// TwinCAT 3 PLC project UnitTests
// Title: tcl_StringUtils_UnitTests
// Company: Red Rock Controls Limited
// Author: Roger Christopher
// ProjectVersion: 1.0.1.0
// Description: Tests tcl_StringUtils V 1.0.5.0 Updated to use tcl_SimpleUnitTestLibrary V1.0.2.0
// ProgramVersion: 3.1.4024.0
// libraries:
//   Tc2_Standard, * (Beckhoff Automation GmbH)
//   Tc2_System, * (Beckhoff Automation GmbH)
//   Tc2_Utilities, * (Beckhoff Automation GmbH)
//   Tc3_Module, * (Beckhoff Automation GmbH)
//   tcl_StringUtils, * (Red Rock Controls Limited)
//   tcl_UnitTestLibrary, * (Red Rock Controls Limited)
// project tree:
//   / PlcTask.TcTTO
//   Unit Tests/ MAIN.TcPOU, T_TestSuite.TcPOU
//   Unit Tests/String Utils/Conversion/ Test_StringToIpAddress.TcPOU
//   Unit Tests/String Utils/Date Time Formatting Tests/ Test_F_DateAsString_ReturnsDateString.TcPOU, Test_F_DateTimeAsString.TcPOU, Test_F_DateTimeAsString_ms.TcPOU, Test_F_TimeAsString_Returns24HourFormat.TcPOU, Test_F_TimeAsString_ReturnsLeadingZeros.TcPOU, Test_F_TimeAsString_ms_ReturnsString_ms.TcPOU, Test_F_TimestampAsFilename_ReturnsValue.TcPOU, Test_F_TimestampAsFilename_ms.TcPOU
//   Unit Tests/String Utils/Format String Tests/ Test_FormatStringWith4CharHexValue.TcPOU, Test_FormatStringWith8CharHexValue.TcPOU, Test_F_PadString_PadsShortStrings.TcPOU, Test_F_PadString_TruncsLongStrings.TcPOU
//   Unit Tests/String Utils/LTrimEx/ Test_LTrimEx_HandlesEmptySubject.TcPOU, Test_LTrimEx_HandlesTrimmingManyChars.TcPOU, Test_LTrimEx_HandlesTrimmingNoChars.TcPOU
//   Unit Tests/String Utils/RTrimEx/ Test_RTrimEx_HandlesEmptySubject.TcPOU, Test_RTrimEx_HandlesTrimmingManyChars.TcPOU, Test_RTrimEx_HandlesTrimmingNoChars.TcPOU
//   Unit Tests/String Utils/String Split/ Test_TStringSplitter_Handles_Empty_String.TcPOU, Test_TStringSplitter_Handles_Empty_SubString.TcPOU, Test_TStringSplitter_Handles_Multiple_Empty.TcPOU, Test_TStringSplitter_ReturnsRemainder.TcPOU, Test_TStringSplitter_Splits_On_Tab.TcPOU
//   Unit Tests/String Utils/Trim/ Test_TrimEx_HandlesEmptySubject.TcPOU, Test_TrimEx_HandlesTrimmingOnlyWhitespace.TcPOU
// (motion and I/O tree: see PLC project tcl_stringutils)
// real-time tasks:
//   TASK PlcTask: cycle T#10ms, priority 1, ADS port 350

CONFIGURATION UnitTests
    RESOURCE PLC ON TwinCAT3
        TASK PlcTask(INTERVAL := T#10ms, PRIORITY := 1);
        PROGRAM MAIN WITH PlcTask : MAIN;
    END_RESOURCE
END_CONFIGURATION

// ---- Unit Tests/MAIN.TcPOU
PROGRAM MAIN
VAR
    TestSuite : T_TestSuite;
END_VAR

TestSuite();

END_PROGRAM

// ---- Unit Tests/T_TestSuite.TcPOU
{attribute 'call_after_init'}
FUNCTION_BLOCK T_TestSuite
VAR
    Test_StringToIpAddress                                 : Test_StringToIpAddress;
    Test_FormatStringWith4CharHexValue                     : Test_FormatStringWith4CharHexValue;
    Test_FormatStringWith8CharHexValue                     : Test_FormatStringWith8CharHexValue;
    Test_LTrimEx_HandlesEmptySubject                       : Test_LTrimEx_HandlesEmptySubject;
    Test_LTrimEx_HandlesTrimmingNoChars                    : Test_LTrimEx_HandlesTrimmingNoChars;
    Test_LTrimEx_HandlesTrimmingManyChars                  : Test_LTrimEx_HandlesTrimmingManyChars;
    Test_RTrimEx_HandlesEmptySubject                       : Test_RTrimEx_HandlesEmptySubject;
    Test_RTrimEx_HandlesTrimmingNoChars                    : Test_RTrimEx_HandlesTrimmingNoChars;
    Test_RTrimEx_HandlesTrimmingManyChars                  : Test_RTrimEx_HandlesTrimmingManyChars;
    Test_TrimEx_HandlesTrimmingOnlyWhitespace              : Test_TrimEx_HandlesTrimmingOnlyWhitespace;
    Test_TrimEx_HandlesEmptySubject                        : Test_TrimEx_HandlesEmptySubject;
    Test_F_DateAsString_ReturnsDateString                  : Test_F_DateAsString_ReturnsDateString;
    Test_F_DateTimeAsString_ReturnsDateTimeString          : Test_F_DateTimeAsString;
    Test_F_DateTimeAsString_ms_ReturnsDTStr                : Test_F_DateTimeAsString_ms;
    Test_F_TimeAsString_Returns24HourFormat                : Test_F_TimeAsString_Returns24HourFormat;
    Test_F_TimeAsString_ReturnsLeadingZeros                : Test_F_TimeAsString_ReturnsLeadingZeros;
    Test_F_TimeAsString_ms_ReturnsTimeString_ms            : Test_F_TimeAsString_ms_ReturnsString_ms;
    Test_F_TimestampAsFilenameString_ReturnsFilenameString : Test_F_TimestampAsFilename_ReturnsValue;
    Test_TStringSplitter_Handles_Empty_String              : Test_TStringSplitter_Handles_Empty_String;
    Test_TStringSplitter_ReturnsRemainder                  : Test_TStringSplitter_ReturnsRemainder;
    Test_TStringSplitter_Splits_On_Tab                     : Test_TStringSplitter_Splits_On_Tab;
    Test_TStringSplitter_Handles_Empty_SubString           : Test_TStringSplitter_Handles_Empty_SubString;
    Test_TStringSplitter_Handles_Multiple_Empty_SubStrings : Test_TStringSplitter_Handles_Multiple_Empty;
    Test_F_PadString_PadsShortStrings                      : Test_F_PadString_PadsShortStrings;
    Test_F_PadString_TruncsLongString                      : Test_F_PadString_TruncsLongStrings;
    Test_F_TimestampAsFilename_ms                          : Test_F_TimestampAsFilename_ms;
END_VAR

Test_StringToIpAddress.RunTest();
Test_FormatStringWith4CharHexValue.RunTest();
Test_FormatStringWith8CharHexValue.RunTest();
Test_LTrimEx_HandlesEmptySubject.RunTest();
Test_LTrimEx_HandlesTrimmingNoChars.RunTest();
Test_LTrimEx_HandlesTrimmingManyChars.RunTest();
Test_RTrimEx_HandlesEmptySubject.RunTest();
Test_RTrimEx_HandlesTrimmingNoChars.RunTest();
Test_RTrimEx_HandlesTrimmingManyChars.RunTest();
Test_TrimEx_HandlesTrimmingOnlyWhitespace.RunTest();
Test_TrimEx_HandlesEmptySubject.RunTest();
Test_F_DateAsString_ReturnsDateString.RunTest();
Test_F_DateTimeAsString_ReturnsDateTimeString.RunTest();
Test_F_DateTimeAsString_ms_ReturnsDTStr.RunTest();
Test_F_TimeAsString_Returns24HourFormat.RunTest();
Test_F_TimeAsString_ReturnsLeadingZeros.RunTest();
Test_F_TimeAsString_ms_ReturnsTimeString_ms.RunTest();
Test_F_TimestampAsFilenameString_ReturnsFilenameString.RunTest();
Test_TStringSplitter_Handles_Empty_String.RunTest();
Test_TStringSplitter_ReturnsRemainder.RunTest();
Test_TStringSplitter_Splits_On_Tab.RunTest();
Test_TStringSplitter_Handles_Empty_SubString.RunTest();
Test_TStringSplitter_Handles_Multiple_Empty_SubStrings.RunTest();
Test_F_PadString_PadsShortStrings.RunTest();
Test_F_PadString_TruncsLongString.RunTest();
Test_F_TimestampAsFilename_ms.RunTest();

END_FUNCTION_BLOCK

// ---- Unit Tests/String Utils/Conversion/Test_StringToIpAddress.TcPOU
FUNCTION_BLOCK Test_StringToIpAddress EXTENDS T_UnitTestBase
VAR
    SubjectString : T_MaxString := '192.168.1.120';
    Result        : ARRAY[1..4] OF BYTE;
END_VAR

{attribute 'analysis' := '-33'} // inhibit unused variable warning
METHOD RunTest
IF Retest THEN
	SUPER^.Init();
END_IF

IF TestCompleted THEN
	RETURN;
END_IF

Result := F_String_To_IPv4_Address(SubjectString);

AssertEquals_BYTE(Expected := 120,
                  Actual   := Result[1],
                  Message  := 'F_String_To_IPv4_Address(SubjectString)');

AssertEquals_BYTE(Expected := 1,
                  Actual   := Result[2],
                  Message  := 'F_String_To_IPv4_Address(SubjectString)');

AssertEquals_BYTE(Expected := 168,
                  Actual   := Result[3],
                  Message  := 'F_String_To_IPv4_Address(SubjectString)');

AssertEquals_BYTE(Expected := 192,
                  Actual   := Result[4],
                  Message  := 'F_String_To_IPv4_Address(SubjectString)');

TestCompleted := TRUE;
END_METHOD

END_FUNCTION_BLOCK

// ---- Unit Tests/String Utils/Format String Tests/Test_FormatStringWith4CharHexValue.TcPOU
FUNCTION_BLOCK Test_FormatStringWith4CharHexValue EXTENDS T_UnitTestBase
VAR_INPUT
END_VAR
VAR_OUTPUT
END_VAR
VAR
    FormattedString : T_MaxString;
    Value           : UINT;
END_VAR

{attribute 'analysis' := '-33'} // inhibit unused variable warning
METHOD RunTest
IF Retest THEN
	SUPER^.Init();
END_IF

IF TestCompleted THEN
	RETURN;
END_IF

Value           := 16#12AB;
FormattedString := F_FormatString1('Hex value = 0x%0.4X', F_UINT(Value));

AssertEquals_STRING(Expected := 'Hex value = 0x12AB',
                    Actual   := FormattedString,
                    Message  := 'FormattedString');

TestCompleted := TRUE;
END_METHOD

END_FUNCTION_BLOCK

// ---- Unit Tests/String Utils/Format String Tests/Test_FormatStringWith8CharHexValue.TcPOU
FUNCTION_BLOCK Test_FormatStringWith8CharHexValue EXTENDS T_UnitTestBase
VAR_INPUT
END_VAR
VAR_OUTPUT
END_VAR
VAR
    FormattedString : T_MaxString;
    Value           : UDINT;
END_VAR

{attribute 'analysis' := '-33'} // inhibit unused variable warning
METHOD RunTest
IF Retest THEN
	SUPER^.Init();
END_IF

IF TestCompleted THEN
	RETURN;
END_IF

Value           := 16#12AB;
FormattedString := F_FormatString1('Hex value = 0x%0.8X', F_UDINT(Value));

AssertEquals_STRING(Expected := 'Hex value = 0x000012AB',
                    Actual   := FormattedString,
                    Message  := 'FormattedString');

TestCompleted := TRUE;
END_METHOD

END_FUNCTION_BLOCK

// ---- Unit Tests/String Utils/LTrimEx/Test_LTrimEx_HandlesEmptySubject.TcPOU
FUNCTION_BLOCK Test_LTrimEx_HandlesEmptySubject EXTENDS T_UnitTestBase
VAR_INPUT
END_VAR
VAR_OUTPUT
END_VAR
VAR
    SubjectString : T_MaxString := '';
END_VAR

{attribute 'analysis' := '-33'} // inhibit unused variable warning
METHOD RunTest
IF Retest THEN
	SUPER^.Init();
END_IF

IF TestCompleted THEN
	RETURN;
END_IF

AssertEquals_STRING(Expected := '',
                    Actual   := F_LTrimEx(n := 1, str := SubjectString),
                    Message  := 'F_LTrimEx(SubjectString)');

TestCompleted := TRUE;
END_METHOD

END_FUNCTION_BLOCK

// ---- Unit Tests/String Utils/LTrimEx/Test_LTrimEx_HandlesTrimmingNoChars.TcPOU
FUNCTION_BLOCK Test_LTrimEx_HandlesTrimmingNoChars EXTENDS T_UnitTestBase
VAR_INPUT
END_VAR
VAR_OUTPUT
END_VAR
VAR
    SubjectString : T_MaxString := 'Badger';
END_VAR

{attribute 'analysis' := '-33'} // inhibit unused variable warning
METHOD RunTest
IF Retest THEN
	SUPER^.Init();
END_IF

IF TestCompleted THEN
	RETURN;
END_IF

AssertEquals_STRING(Expected := 'Badger',
                    Actual   := F_LTrimEx(n := 0, str := SubjectString),
                    Message  := 'F_LTrimEx(SubjectString)');

TestCompleted := TRUE;
END_METHOD

END_FUNCTION_BLOCK

// ---- Unit Tests/String Utils/LTrimEx/Test_LTrimEx_HandlesTrimmingManyChars.TcPOU
FUNCTION_BLOCK Test_LTrimEx_HandlesTrimmingManyChars EXTENDS T_UnitTestBase
VAR_INPUT
END_VAR
VAR_OUTPUT
END_VAR
VAR
    SubjectString : T_MaxString := 'Badger';
END_VAR

{attribute 'analysis' := '-33'} // inhibit unused variable warning
METHOD RunTest
IF Retest THEN
	SUPER^.Init();
END_IF

IF TestCompleted THEN
	RETURN;
END_IF

AssertEquals_STRING(Expected := '',
                    Actual   := F_LTrimEx(n := 20, str := SubjectString),
                    Message  := 'F_LTrimEx(SubjectString)');

TestCompleted := TRUE;
END_METHOD

END_FUNCTION_BLOCK

// ---- Unit Tests/String Utils/RTrimEx/Test_RTrimEx_HandlesEmptySubject.TcPOU
FUNCTION_BLOCK Test_RTrimEx_HandlesEmptySubject EXTENDS T_UnitTestBase
VAR_INPUT
END_VAR
VAR_OUTPUT
END_VAR
VAR
    SubjectString : T_MaxString := '';
END_VAR

{attribute 'analysis' := '-33'} // inhibit unused variable warning
METHOD RunTest
IF Retest THEN
	SUPER^.Init();
END_IF

IF TestCompleted THEN
	RETURN;
END_IF

AssertEquals_STRING(Expected := '',
                    Actual   := F_RTrimEx(n := 1, str := SubjectString),
                    Message  := 'F_LTrimEx(SubjectString)');

TestCompleted := TRUE;
END_METHOD

END_FUNCTION_BLOCK

// ---- Unit Tests/String Utils/RTrimEx/Test_RTrimEx_HandlesTrimmingNoChars.TcPOU
FUNCTION_BLOCK Test_RTrimEx_HandlesTrimmingNoChars EXTENDS T_UnitTestBase
VAR_INPUT
END_VAR
VAR_OUTPUT
END_VAR
VAR
    SubjectString : T_MaxString := 'Badger';
END_VAR

{attribute 'analysis' := '-33'} // inhibit unused variable warning
METHOD RunTest
IF Retest THEN
	SUPER^.Init();
END_IF

IF TestCompleted THEN
	RETURN;
END_IF

AssertEquals_STRING(Expected := 'Badger',
                    Actual   := F_RTrimEx(n := 0, str := SubjectString),
                    Message  := 'F_LTrimEx(SubjectString)');

TestCompleted := TRUE;
END_METHOD

END_FUNCTION_BLOCK

// ---- Unit Tests/String Utils/RTrimEx/Test_RTrimEx_HandlesTrimmingManyChars.TcPOU
FUNCTION_BLOCK Test_RTrimEx_HandlesTrimmingManyChars EXTENDS T_UnitTestBase
VAR_INPUT
END_VAR
VAR_OUTPUT
END_VAR
VAR
    SubjectString : T_MaxString := 'Badger';
END_VAR

{attribute 'analysis' := '-33'} // inhibit unused variable warning
METHOD RunTest
IF Retest THEN
	SUPER^.Init();
END_IF

IF TestCompleted THEN
	RETURN;
END_IF

AssertEquals_STRING(Expected := '',
                    Actual   := F_RTrimEx(n := 20, str := SubjectString),
                    Message  := 'F_LTrimEx(SubjectString)');

TestCompleted := TRUE;
END_METHOD

END_FUNCTION_BLOCK

// ---- Unit Tests/String Utils/Trim/Test_TrimEx_HandlesTrimmingOnlyWhitespace.TcPOU
FUNCTION_BLOCK Test_TrimEx_HandlesTrimmingOnlyWhitespace EXTENDS T_UnitTestBase
VAR_INPUT
END_VAR
VAR_OUTPUT
END_VAR
VAR
    SubjectString : T_MaxString := '$T$T$T$T$T$R$R    $R';
END_VAR

{attribute 'analysis' := '-33'} // inhibit unused variable warning
METHOD RunTest
IF Retest THEN
	SUPER^.Init();
END_IF

IF TestCompleted THEN
	RETURN;
END_IF

AssertEquals_STRING(Expected := '',
                    Actual   := F_Trim(str := SubjectString),
                    Message  := 'F_LTrimEx(SubjectString)');

TestCompleted := TRUE;
END_METHOD

END_FUNCTION_BLOCK

// ---- Unit Tests/String Utils/Trim/Test_TrimEx_HandlesEmptySubject.TcPOU
FUNCTION_BLOCK Test_TrimEx_HandlesEmptySubject EXTENDS T_UnitTestBase
VAR_INPUT
END_VAR
VAR_OUTPUT
END_VAR
VAR
    SubjectString : T_MaxString := '';
END_VAR

{attribute 'analysis' := '-33'} // inhibit unused variable warning
METHOD RunTest
IF Retest THEN
	SUPER^.Init();
END_IF

IF TestCompleted THEN
	RETURN;
END_IF

AssertEquals_STRING(Expected := '',
                    Actual   := F_Trim(str := SubjectString),
                    Message  := 'F_Trim(str := SubjectString)');

TestCompleted := TRUE;
END_METHOD

END_FUNCTION_BLOCK

// ---- Unit Tests/String Utils/Date Time Formatting Tests/Test_F_DateAsString_ReturnsDateString.TcPOU
FUNCTION_BLOCK Test_F_DateAsString_ReturnsDateString EXTENDS T_UnitTestBase
VAR
    TimeStruct : TIMESTRUCT := (wDay := 23, wMonth := 12, wYear := 1945);
END_VAR

{attribute 'analysis' := '-33'} // inhibit unused variable warning
METHOD RunTest
IF Retest THEN
	SUPER^.Init();
END_IF

IF TestCompleted THEN
	RETURN;
END_IF

AssertEquals_STRING(Expected := '23/12/1945',
                    Actual   := F_DateAsString(TimeStruct),
                    Message  := 'F_DateAsString(TimeStruct)');

TestCompleted := TRUE;
END_METHOD

END_FUNCTION_BLOCK

// ---- Unit Tests/String Utils/Date Time Formatting Tests/Test_F_DateTimeAsString.TcPOU
FUNCTION_BLOCK Test_F_DateTimeAsString EXTENDS T_UnitTestBase
VAR
    TimeStruct : TIMESTRUCT := (wDay    := 23,
                                wMonth  := 12,
                                wYear   := 1945,
                                wHour   := 22,
                                wMinute := 20,
                                wSecond := 18);
END_VAR

{attribute 'analysis' := '-33'} // inhibit unused variable warning
METHOD RunTest
IF Retest THEN
	SUPER^.Init();
END_IF

IF TestCompleted THEN
	RETURN;
END_IF

AssertEquals_STRING(Expected := '22:20:18 23/12/1945',
                    Actual   := F_DateTimeAsString(TimeStruct),
                    Message  := 'F_DateTimeAsString(TimeStruct)');

TestCompleted := TRUE;
END_METHOD

END_FUNCTION_BLOCK

// ---- Unit Tests/String Utils/Date Time Formatting Tests/Test_F_DateTimeAsString_ms.TcPOU
FUNCTION_BLOCK Test_F_DateTimeAsString_ms EXTENDS T_UnitTestBase
VAR
    TimeStruct : TIMESTRUCT := (wDay          := 23,
                                wMonth        := 12,
                                wYear         := 1945,
                                wHour         := 22,
                                wMinute       := 20,
                                wSecond       := 18,
                                wMilliseconds := 512);
END_VAR

{attribute 'analysis' := '-33'} // inhibit unused variable warning
METHOD RunTest
IF Retest THEN
	SUPER^.Init();
END_IF

IF TestCompleted THEN
	RETURN;
END_IF

AssertEquals_STRING(Expected := '22:20:18.512 23/12/1945',
                    Actual   := F_DateTimeAsString_ms(TimeStruct),
                    Message  := 'F_DateTimeAsString_ms(TimeStruct)');

TestCompleted := TRUE;
END_METHOD

END_FUNCTION_BLOCK

// ---- Unit Tests/String Utils/Date Time Formatting Tests/Test_F_TimeAsString_Returns24HourFormat.TcPOU
FUNCTION_BLOCK Test_F_TimeAsString_Returns24HourFormat EXTENDS T_UnitTestBase
VAR
    TimeStruct : TIMESTRUCT := (wHour := 22, wMinute := 20, wSecond := 18);
END_VAR

{attribute 'analysis' := '-33'} // inhibit unused variable warning
METHOD RunTest
IF Retest THEN
	SUPER^.Init();
END_IF

IF TestCompleted THEN
	RETURN;
END_IF

AssertEquals_STRING(Expected := '22:20:18',
                    Actual   := F_TimeAsString(TimeStruct),
                    Message  := 'F_TimeAsString(TimeStruct)');

TestCompleted := TRUE;
END_METHOD

END_FUNCTION_BLOCK

// ---- Unit Tests/String Utils/Date Time Formatting Tests/Test_F_TimeAsString_ReturnsLeadingZeros.TcPOU
FUNCTION_BLOCK Test_F_TimeAsString_ReturnsLeadingZeros EXTENDS T_UnitTestBase
VAR
    TimeStruct : TIMESTRUCT := (wHour := 6, wMinute := 5, wSecond := 4);
END_VAR

{attribute 'analysis' := '-33'} // inhibit unused variable warning
METHOD RunTest
IF Retest THEN
	SUPER^.Init();
END_IF

IF TestCompleted THEN
	RETURN;
END_IF

AssertEquals_STRING(Expected := '06:05:04',
                    Actual   := F_TimeAsString(TimeStruct),
                    Message  := 'F_TimeAsString(TimeStruct)');

TestCompleted := TRUE;
END_METHOD

END_FUNCTION_BLOCK

// ---- Unit Tests/String Utils/Date Time Formatting Tests/Test_F_TimeAsString_ms_ReturnsString_ms.TcPOU
FUNCTION_BLOCK Test_F_TimeAsString_ms_ReturnsString_ms EXTENDS T_UnitTestBase
VAR
    TimeStruct : TIMESTRUCT := (wHour := 6, wMinute := 5, wSecond := 4, wMilliseconds := 135);
END_VAR

{attribute 'analysis' := '-33'} // inhibit unused variable warning
METHOD RunTest
IF Retest THEN
	SUPER^.Init();
END_IF

IF TestCompleted THEN
	RETURN;
END_IF

AssertEquals_STRING(Expected := '06:05:04.135',
                    Actual   := F_TimeAsString_ms(TimeStruct),
                    Message  := 'F_TimeAsString_ms(TimeStruct)');

TestCompleted := TRUE;
END_METHOD

END_FUNCTION_BLOCK

// ---- Unit Tests/String Utils/Date Time Formatting Tests/Test_F_TimestampAsFilename_ReturnsValue.TcPOU
FUNCTION_BLOCK Test_F_TimestampAsFilename_ReturnsValue EXTENDS T_UnitTestBase
VAR
    TimeStruct : TIMESTRUCT := (wDay          := 23,
                                wMonth        := 12,
                                wYear         := 1945,
                                wHour         := 22,
                                wMinute       := 20,
                                wSecond       := 18,
                                wMilliseconds := 512);
END_VAR

METHOD Init
VAR_INPUT
END_VAR
END_METHOD

{attribute 'analysis' := '-33'} // inhibit unused variable warning
METHOD RunTest
AssertEquals_STRING(Expected := '1945-12-23 22-20-18',
                    Actual   := F_TimestampAsFilenameString(TimeStruct),
                    Message  := 'F_TimeAsString_ms(TimeStruct)');

TestCompleted := TRUE;
END_METHOD

END_FUNCTION_BLOCK

// ---- Unit Tests/String Utils/String Split/Test_TStringSplitter_Handles_Empty_String.TcPOU
FUNCTION_BLOCK Test_TStringSplitter_Handles_Empty_String EXTENDS T_UnitTestBase
VAR
    StringSplitter : T_StringSplitter;
END_VAR

{attribute 'analysis' := '-33'} // inhibit unused variable warning
METHOD RunTest
IF Retest THEN
	SUPER^.Init();
END_IF

IF TestCompleted THEN
	RETURN;
END_IF


StringSplitter.Init(Str    := '',
                    Delim1 := '$T',
                    Delim2 := '');

AssertEquals_STRING(Expected := '',
                    Actual   := StringSplitter.GetNext(),
                    Message  := 'StringSplitter.GetNext()');

AssertEquals_BOOL(Expected := FALSE,
                  Actual   := StringSplitter.HasMore(),
                  Message  := 'StringSplitter.HasMore()');

TestCompleted := TRUE;
END_METHOD

END_FUNCTION_BLOCK

// ---- Unit Tests/String Utils/String Split/Test_TStringSplitter_ReturnsRemainder.TcPOU
FUNCTION_BLOCK Test_TStringSplitter_ReturnsRemainder EXTENDS T_UnitTestBase
VAR
    StringSplitter : T_StringSplitter;
END_VAR

{attribute 'analysis' := '-33'} // inhibit unused variable warning
METHOD RunTest
IF Retest THEN
	SUPER^.Init();
END_IF

IF TestCompleted THEN
	RETURN;
END_IF


StringSplitter.Init(Str    := 'Bob$TCharles$TDavid',
                    Delim1 := '$T',
                    Delim2 := '');

AssertEquals_BOOL(Expected := TRUE,
                  Actual   := StringSplitter.HasMore(),
                  Message  := 'StringSplitter.HasMore()');

AssertEquals_STRING(Expected := 'Bob',
                    Actual   := StringSplitter.GetNext(),
                    Message  := 'StringSplitter.GetNext()');

AssertEquals_STRING(Expected := 'Charles$TDavid',
                    Actual   := StringSplitter.GetRemainder(),
                    Message  := 'StringSplitter.GetRemainder()');

AssertEquals_STRING(Expected := '',
                    Actual   := StringSplitter.GetRemainder(),
                    Message  := 'StringSplitter.GetRemainder()');

AssertEquals_BOOL(Expected := FALSE,
                  Actual   := StringSplitter.HasMore(),
                  Message  := 'StringSplitter.HasMore()');

TestCompleted := TRUE;
END_METHOD

END_FUNCTION_BLOCK

// ---- Unit Tests/String Utils/String Split/Test_TStringSplitter_Splits_On_Tab.TcPOU
FUNCTION_BLOCK Test_TStringSplitter_Splits_On_Tab EXTENDS T_UnitTestBase
VAR
    StringSplitter : T_StringSplitter;
END_VAR

{attribute 'analysis' := '-33'} // inhibit unused variable warning
METHOD RunTest
IF Retest THEN
	SUPER^.Init();
END_IF

IF TestCompleted THEN
	RETURN;
END_IF


StringSplitter.Init(Str    := 'Bob$TCharles$TDavid',
                    Delim1 := '$T',
                    Delim2 := '');

AssertEquals_STRING(Expected := 'Bob',
                    Actual   := StringSplitter.GetNext(),
                    Message  := 'StringSplitter.GetNext()');

AssertEquals_STRING(Expected := 'Charles',
                    Actual   := StringSplitter.GetNext(),
                    Message  := 'StringSplitter.GetNext()');

AssertEquals_STRING(Expected := 'David',
                    Actual   := StringSplitter.GetNext(),
                    Message  := 'StringSplitter.GetNext()');

TestCompleted := TRUE;
END_METHOD

END_FUNCTION_BLOCK

// ---- Unit Tests/String Utils/String Split/Test_TStringSplitter_Handles_Empty_SubString.TcPOU
FUNCTION_BLOCK Test_TStringSplitter_Handles_Empty_SubString EXTENDS T_UnitTestBase
VAR
    StringSplitter : T_StringSplitter;
    SubjectString  : T_MaxString := 'Badger,';
END_VAR

{attribute 'analysis' := '-33'} // inhibit unused variable warning
METHOD RunTest
IF Retest THEN
	SUPER^.Init();
END_IF

IF TestCompleted THEN
	RETURN;
END_IF

StringSplitter.Init(Str    := SubjectString,
                    Delim1 := ',',
                    Delim2 := '');

AssertEquals_STRING(Expected := 'Badger',
                    Actual   := StringSplitter.GetNext(),
                    Message  := 'StringSplitter.GetNext()');

AssertEquals_BOOL(Expected := FALSE,
                  Actual   := StringSplitter.HasMore(),
                  Message  := 'StringSplitter.HasMore()');

AssertEquals_STRING(Expected := '',
                    Actual   := StringSplitter.GetNext(),
                    Message  := 'StringSplitter.GetNext()');

TestCompleted := TRUE;
END_METHOD

END_FUNCTION_BLOCK

// ---- Unit Tests/String Utils/String Split/Test_TStringSplitter_Handles_Multiple_Empty.TcPOU
FUNCTION_BLOCK Test_TStringSplitter_Handles_Multiple_Empty EXTENDS T_UnitTestBase
VAR
    StringSplitter : T_StringSplitter;
    SubjectString  : T_MaxString := 'Badger,,,';
END_VAR

{attribute 'analysis' := '-33'} // inhibit unused variable warning
METHOD RunTest
IF Retest THEN
	SUPER^.Init();
END_IF

IF TestCompleted THEN
	RETURN;
END_IF

StringSplitter.Init(Str    := SubjectString,
                    Delim1 := ',',
                    Delim2 := '');

AssertEquals_STRING(Expected := 'Badger',
                    Actual   := StringSplitter.GetNext(),
                    Message  := 'StringSplitter.GetNext()');

AssertEquals_BOOL(Expected := TRUE,
                  Actual   := StringSplitter.HasMore(),
                  Message  := 'StringSplitter.HasMore()');

AssertEquals_STRING(Expected := '',
                    Actual   := StringSplitter.GetNext(),
                    Message  := 'StringSplitter.GetNext()');

AssertEquals_BOOL(Expected := TRUE,
                  Actual   := StringSplitter.HasMore(),
                  Message  := 'StringSplitter.HasMore()');

AssertEquals_STRING(Expected := '',
                    Actual   := StringSplitter.GetNext(),
                    Message  := 'StringSplitter.GetNext()');

AssertEquals_BOOL(Expected := FALSE,
                  Actual   := StringSplitter.HasMore(),
                  Message  := 'StringSplitter.HasMore()');

TestCompleted := TRUE;
END_METHOD

END_FUNCTION_BLOCK

// ---- Unit Tests/String Utils/Format String Tests/Test_F_PadString_PadsShortStrings.TcPOU
FUNCTION_BLOCK Test_F_PadString_PadsShortStrings EXTENDS T_UnitTestBase
VAR
    SubjectString : T_MaxString;
    ResultString  : T_MaxString;
END_VAR

{attribute 'analysis' := '-33'} // inhibit unused variable warning
METHOD RunTest
IF Retest THEN
	SUPER^.Init();
END_IF

IF TestCompleted THEN
	RETURN;
END_IF

SubjectString := 'Bob';
ResultString  := F_PadString(InputString := SubjectString,
                             Length      := 20);

AssertEquals_INT(Expected := 20,
                 Actual   := LEN(ResultString),
                 Message  := 'LEN(ResultString)');

AssertEquals_STRING(Expected := 'Bob                 ',
                    Actual   := ResultString,
                    Message  := 'ResultString');

TestCompleted := TRUE;
END_METHOD

END_FUNCTION_BLOCK

// ---- Unit Tests/String Utils/Format String Tests/Test_F_PadString_TruncsLongStrings.TcPOU
FUNCTION_BLOCK Test_F_PadString_TruncsLongStrings EXTENDS T_UnitTestBase
VAR
    SubjectString : T_MaxString;
    ResultString  : T_MaxString;
END_VAR

{attribute 'analysis' := '-33'} // inhibit unused variable warning
METHOD RunTest
IF Retest THEN
	SUPER^.Init();
END_IF

IF TestCompleted THEN
	RETURN;
END_IF

SubjectString := 'A long message with too many characters';
ResultString  := F_PadString(InputString := SubjectString,
                             Length      := 20);

AssertEquals_INT(Expected := 20,
                 Actual   := LEN(ResultString),
                 Message  := 'LEN(ResultString)');

AssertEquals_STRING(Expected := 'A long message with ',
                    Actual   := ResultString,
                    Message  := 'ResultString');

TestCompleted := TRUE;
END_METHOD

END_FUNCTION_BLOCK

// ---- Unit Tests/String Utils/Date Time Formatting Tests/Test_F_TimestampAsFilename_ms.TcPOU
FUNCTION_BLOCK Test_F_TimestampAsFilename_ms EXTENDS T_UnitTestBase
VAR
    TimeStruct : TIMESTRUCT := (wDay          := 23,
                                wMonth        := 12,
                                wYear         := 1945,
                                wHour         := 22,
                                wMinute       := 20,
                                wSecond       := 18,
                                wMilliseconds := 512);
END_VAR

{attribute 'analysis' := '-33'} // inhibit unused variable warning
METHOD RunTest
IF Retest THEN
	SUPER^.Init();
END_IF

IF TestCompleted THEN
	RETURN;
END_IF

AssertEquals_STRING(Expected := '1945-12-23 22:20:18.512',
                    Actual   := F_TimestampAsFilenameString_ms(TimeStruct),
                    Message  := 'F_TimestampAsFilenameString_ms(TimeStruct)');

TestCompleted := TRUE;
END_METHOD

END_FUNCTION_BLOCK
